PROGRAM Main
VAR
  counter : INT := 0;
  bEnable : BOOL;
END_VAR

IF bEnable THEN
  counter := counter + 1;
END_IF

END_PROGRAM

(* stored: Version 1.1.0.1
   POU Main: Id {00000000-0000-0000-0000-000000000001}, SpecialFunc None *)
